{attribute 'linkalways'} 
{attribute 'no_explicit_call' := 'This FB is a CLASS and must be accessed using methods or properties'}
{attribute 'enable_dynamic_creation'}
FUNCTION_BLOCK Node_F_VN_AddImagesWeighted EXTENDS VisionNode
VAR
    ipSrcImage1 : _ITcVnImage;
    ipSrcImage2 : _ITcVnImage;
    ipDestImage : _ITcVnImage;
    fWeight1 : _LREAL(0.0);
    fWeight2 : _LREAL(0.0);
    fDelta : _LREAL(0.0);
    hrPrev : _HRESULT(S_OK);
	hresult : _HRESULT(S_OK);
END_VAR

METHOD PUBLIC  Clone : I_Node
VAR
	pNode : POINTER TO Node_F_VN_AddImagesWeighted;
END_VAR
pNode := __NEW(Node_F_VN_AddImagesWeighted);
Clone := pNode^;
END_METHOD

METHOD FB_init : BOOL
VAR_INPUT
	bInitRetains : BOOL; // if TRUE, the retain variables are initialized (warm start / cold start)
	bInCopyCode : BOOL;  // if TRUE, the instance afterwards gets moved into the copy code (online change)
END_VAR
AddInput('ipSrcImage1', ipSrcImage1);
AddInput('ipSrcImage2', ipSrcImage2);
AddInput('hrPrev', hrPrev);
AddParameter('fWeight1', fWeight1);
AddParameter('fWeight2', fWeight2);
AddParameter('fDelta', fDelta);
AddOutput('ipDestImage', ipDestImage);
AddOutput('hresult',hresult);
END_METHOD

METHOD PROTECTED OnExecute : HRESULT
hresult.Value := F_VN_AddImagesWeighted(
    ipSrcImage1 := ipSrcImage1.Value,
    ipSrcImage2 := ipSrcImage2.Value,
	ipDestImage := ipDestImage.Value,
    fWeight1 := fWeight1.Value,
    fWeight2 := fWeight2.Value,
    fDelta := fDelta.Value,
	hrPrev:= hrPrev.Value);
END_METHOD

METHOD PUBLIC PreExecutionCheck
VAR_INPUT
	Check : I_PreExecutionChecks;
END_VAR
IF FAILED(hrPrev.Value) THEN
    RETURN;
END_IF

Check.IsTrue(ipSrcImage1.IsValid, 'ipSrcImage1 must contain an image');
Check.IsTrue(ipSrcImage2.IsValid, 'ipSrcImage2 must contain an image');
END_METHOD

END_FUNCTION_BLOCK

(* stored: Version 1.1.0.1, ProductVersion 3.1.4024.13
   POU Node_F_VN_AddImagesWeighted: Id {2477f390-fdc5-057b-25e0-637b3d7869d9}, SpecialFunc None
   Folder Constructor: Id {11f15d47-2146-0209-0d01-3efb1746e51f}
   Method Clone: Id {29e505b4-729c-0107-1d5e-041fce28d8de}
   Method FB_init: Id {b47fc04e-fcb8-0f7b-306f-13ddae238bbd}
   Method OnExecute: Id {2dd81967-e36c-061d-2ff4-6d423e5f292a}
   Method PreExecutionCheck: Id {d7fc67f7-0d4a-0f1d-3090-bc135fe05533} *)
